// TIA Portal V17 export
// export: Created 2026-04-13T11:12:52.5177813Z, ExportSetting WithDefaults, DisplayName Totally Integrated Automation Portal, DisplayVersion V17 Update 4, DisplayName TIA Portal Openness, DisplayVersion V17 Update 4, DisplayName TIA Portal Version Control Interface, DisplayVersion V17, DisplayName SINAMICS Startdrive Advanced, DisplayVersion V17, DisplayName SINAMICS Startdrive G130, G150, S120, S150, SINAMICS MV, S210, DisplayVersion V17, DisplayName SINAMICS Startdrive G110M, G120, G120C, G120D, G120P, G115D, DisplayVersion V17, DisplayName STEP 7 Professional, DisplayVersion V17 Update 4, DisplayName STEP 7 Safety, DisplayVersion V17, DisplayName WinCC Professional, DisplayVersion V17 Update 4
TagTable "OUTCIPCS"
  OUTCIPCS_1设定时间 : Real  (PLC tag OUTCIPCS.1设定时间, HMI_连接_1, 1 s)
  OUTCIPCS_2设定时间 : Real  (PLC tag OUTCIPCS.2设定时间, HMI_连接_1, 1 s)
  OUTCIPCS_3设定时间 : Real  (PLC tag OUTCIPCS.3设定时间, HMI_连接_1, 1 s)
  OUTCIPCS_4设定时间 : Real  (PLC tag OUTCIPCS.4设定时间, HMI_连接_1, 1 s)
  OUTCIPCS_5设定时间 : Real  (PLC tag OUTCIPCS.5设定时间, HMI_连接_1, 1 s)
  OUTCIPCS_6设定时间 : Real  (PLC tag OUTCIPCS.6设定时间, HMI_连接_1, 1 s)
  OUTCIPCS_7设定时间 : Real  (PLC tag OUTCIPCS.7设定时间, HMI_连接_1, 1 s)
  OUTCIPCS_8设定时间 : Real  (PLC tag OUTCIPCS.8设定时间, HMI_连接_1, 1 s)
  OUTCIPCS_9设定时间 : Real  (PLC tag OUTCIPCS.9设定时间, HMI_连接_1, 1 s)
  OUTCIPCS_10设定时间 : Real  (PLC tag OUTCIPCS.10设定时间, HMI_连接_1, 1 s)
  OUTCIPCS_11设定时间 : Real  (PLC tag OUTCIPCS.11设定时间, HMI_连接_1, 1 s)
  OUTCIPCS_12设定时间 : Real  (PLC tag OUTCIPCS.12设定时间, HMI_连接_1, 1 s)
  OUTCIPCS_13设定时间 : Real  (PLC tag OUTCIPCS.13设定时间, HMI_连接_1, 1 s)
  OUTCIPCS_14设定时间 : Real  (PLC tag OUTCIPCS.14设定时间, HMI_连接_1, 1 s)
  OUTCIPCS_15设定时间 : Real  (PLC tag OUTCIPCS.15设定时间, HMI_连接_1, 1 s)
  OUTCIPCS_16设定时间 : Real  (PLC tag OUTCIPCS.16设定时间, HMI_连接_1, 1 s)
  OUTCIPCS_0计时 : Real  (PLC tag OUTCIPCS.0计时, HMI_连接_1, 1 s)
  OUTCIPCS_1计时 : Real  (PLC tag OUTCIPCS.1计时, HMI_连接_1, 1 s)
  OUTCIPCS_2计时 : Real  (PLC tag OUTCIPCS.2计时, HMI_连接_1, 1 s)
  OUTCIPCS_3计时 : Real  (PLC tag OUTCIPCS.3计时, HMI_连接_1, 1 s)
  OUTCIPCS_4计时 : Real  (PLC tag OUTCIPCS.4计时, HMI_连接_1, 1 s)
  OUTCIPCS_5计时 : Real  (PLC tag OUTCIPCS.5计时, HMI_连接_1, 1 s)
  OUTCIPCS_6计时 : Real  (PLC tag OUTCIPCS.6计时, HMI_连接_1, 1 s)
  OUTCIPCS_7计时 : Real  (PLC tag OUTCIPCS.7计时, HMI_连接_1, 1 s)
  OUTCIPCS_8计时 : Real  (PLC tag OUTCIPCS.8计时, HMI_连接_1, 1 s)
  OUTCIPCS_9计时 : Real  (PLC tag OUTCIPCS.9计时, HMI_连接_1, 1 s)
  OUTCIPCS_10计时 : Real  (PLC tag OUTCIPCS.10计时, HMI_连接_1, 1 s)
  OUTCIPCS_11计时 : Real  (PLC tag OUTCIPCS.11计时, HMI_连接_1, 1 s)
  OUTCIPCS_12计时 : Real  (PLC tag OUTCIPCS.12计时, HMI_连接_1, 1 s)
  OUTCIPCS_13计时 : Real  (PLC tag OUTCIPCS.13计时, HMI_连接_1, 1 s)
  OUTCIPCS_14计时 : Real  (PLC tag OUTCIPCS.14计时, HMI_连接_1, 1 s)
  OUTCIPCS_15计时 : Real  (PLC tag OUTCIPCS.15计时, HMI_连接_1, 1 s)
  OUTCIPCS_16计时 : Real  (PLC tag OUTCIPCS.16计时, HMI_连接_1, 1 s)
